// SIMATIC S7-200 project (STEP 7-Micro/WIN), CPU 221 REL 01.10

SYMBOL_TABLE USER1
chay             I0.0
Xanh             Q1.6
Do               Q2.0
Vang             Q2.2
dung             I0.1
END_SYMBOL_TABLE

ORGANIZATION_BLOCK MAIN:OB1
TITLE=PROGRAM COMMENTS
BEGIN
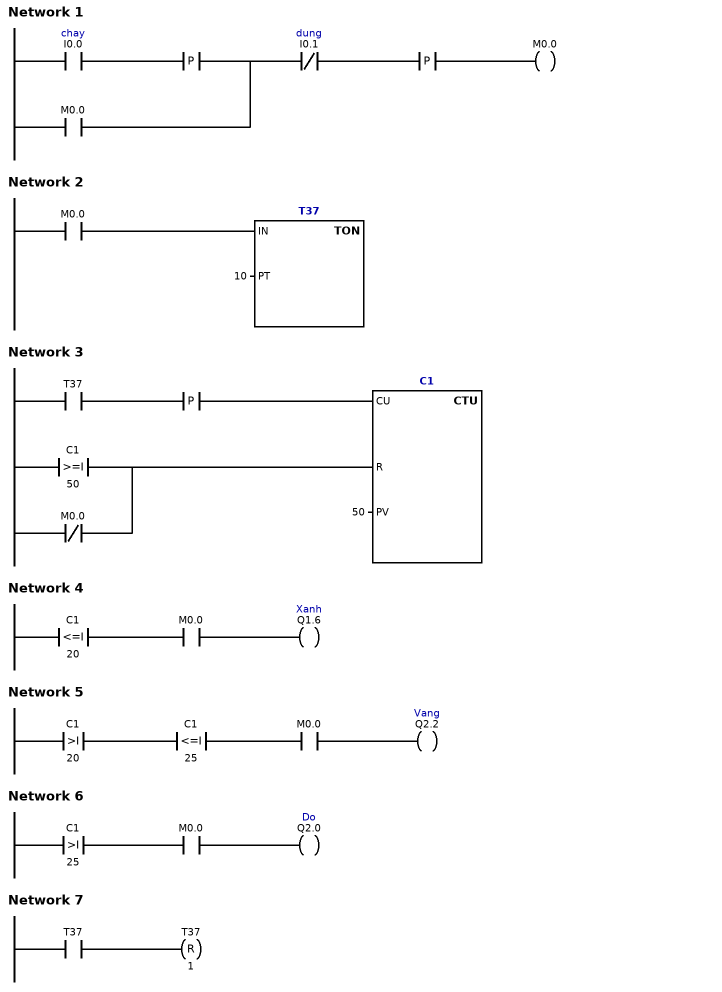
Network 1
LD     chay:I0.0
EU
O      M0.0
AN     dung:I0.1
EU
=      M0.0
Network 2
LD     M0.0
TON    T37, 10
Network 3
LD     T37
EU
LDW>=  C1, 50
ON     M0.0
CTU    C1, 50
Network 4
LDW<=  C1, 20
A      M0.0
=      Xanh:Q1.6
Network 5
LDW>   C1, 20
AW<=   C1, 25
A      M0.0
=      Vang:Q2.2
Network 6
LDW>   C1, 25
A      M0.0
=      Do:Q2.0
Network 7
LD     T37
R      T37, 1
END_ORGANIZATION_BLOCK
